{attribute 'linkalways'} 
{attribute 'no_explicit_call' := 'This FB is a CLASS and must be accessed using methods or properties'}
{attribute 'enable_dynamic_creation'}
FUNCTION_BLOCK Node_F_VN_AddToContainerElements_TcVnVector2_SINT EXTENDS VisionNode
VAR
    aValue : _TcVnVector2_SINT;
    ipContainer : _ITcVnContainer;
    hrPrev : _HRESULT(S_OK);
    hresult : _HRESULT(S_OK);
END_VAR

METHOD PUBLIC  Clone : I_Node
VAR
    pNode : POINTER TO Node_F_VN_AddToContainerElements_TcVnVector2_SINT;
END_VAR
pNode := __NEW(Node_F_VN_AddToContainerElements_TcVnVector2_SINT);
Clone := pNode^;
END_METHOD

METHOD FB_init : BOOL
VAR_INPUT
    bInitRetains : BOOL; // if TRUE, the retain variables are initialized (warm start / cold start)
    bInCopyCode : BOOL;  // if TRUE, the instance afterwards gets moved into the copy code (online change)
END_VAR
AddInput('aValue', aValue);
AddInput('ipContainer', ipContainer);
AddInput('hrPrev', hrPrev);
AddOutput('ipContainer', ipContainer);
AddOutput('hresult',hresult);
END_METHOD

METHOD PROTECTED OnExecute : HRESULT
hresult.Value := F_VN_AddToContainerElements_TcVnVector2_SINT(
    aValue := aValue.Value,
    ipContainer := ipContainer.Value,
    hrPrev:= hrPrev.Value);
END_METHOD

METHOD PUBLIC PreExecutionCheck
VAR_INPUT
    Check : I_PreExecutionChecks;
END_VAR
Check.IsTrue(ipContainer.IsValid, 'ipContainer must be a valid container');
Check.IsTrue(ipContainer.HasType(TC_GLOBAL_CONST_LIST.ContainerType_Vector_TcVnVector2_SINT), 'ipContainer contains incorrect type');
END_METHOD

END_FUNCTION_BLOCK

(* stored: Version 1.1.0.1, ProductVersion 3.1.4024.13
   POU Node_F_VN_AddToContainerElements_TcVnVector2_SINT: Id {2f171236-91fb-4d98-8477-6e809a1c90af}, SpecialFunc None
   Folder Constructor: Id {298d1b2c-c48d-4190-be32-f36d1a56d938}
   Method Clone: Id {aa300eb3-bd68-4586-b982-b1df31534403}
   Method FB_init: Id {20e9396e-3aaf-48ac-a3d4-2a3e649556f7}
   Method OnExecute: Id {541e5e16-b656-47c7-9d7a-39ba3927e569}
   Method PreExecutionCheck: Id {358b1e98-0850-497e-9b82-66a6fb427bb8} *)
